(* LS Electric XG5000 project: 04_Practice3 *)
(* PLC LSPLC *)
(* module base 0 slot 0: 입력 모듈:XGI-D21A (DC 24V 입력, 8점 (전류소스/싱크입력)) *)
(* module base 0 slot 1: 출력 모듈:XGQ-RY1A (릴레이 출력, 8점 (2A용, 단독 COM.)) *)

PROGRAM NewProgram (* task: 스캔 프로그램 *)
VAR
    P1 AT %IX0.0.0 : BOOL;
    P1자가유지 AT %MX0 : BOOL;
    P2 AT %IX0.0.1 : BOOL;
    P2자가유지 AT %MX1 : BOOL;
    P3 AT %IX0.0.2 : BOOL;
    P40 AT %QX0.1.0 : BOOL;
    P41 AT %QX0.1.1 : BOOL;
END_VAR

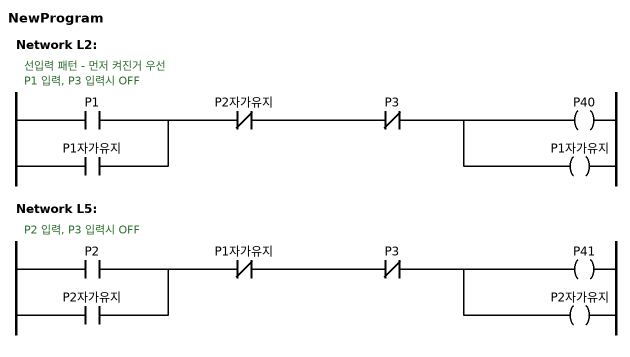
(* 선입력 패턴 - 먼저 켜진거 우선 *)
(* P1 입력, P3 입력시 OFF *)
(* Rung L2 *)
P40 := (P1 OR P1자가유지) AND NOT P2자가유지 AND NOT P3;
P1자가유지 := (P1 OR P1자가유지) AND NOT P2자가유지 AND NOT P3;
(* P2 입력, P3 입력시 OFF *)
(* Rung L5 *)
P41 := (P2 OR P2자가유지) AND NOT P1자가유지 AND NOT P3;
P2자가유지 := (P2 OR P2자가유지) AND NOT P1자가유지 AND NOT P3;
END_PROGRAM